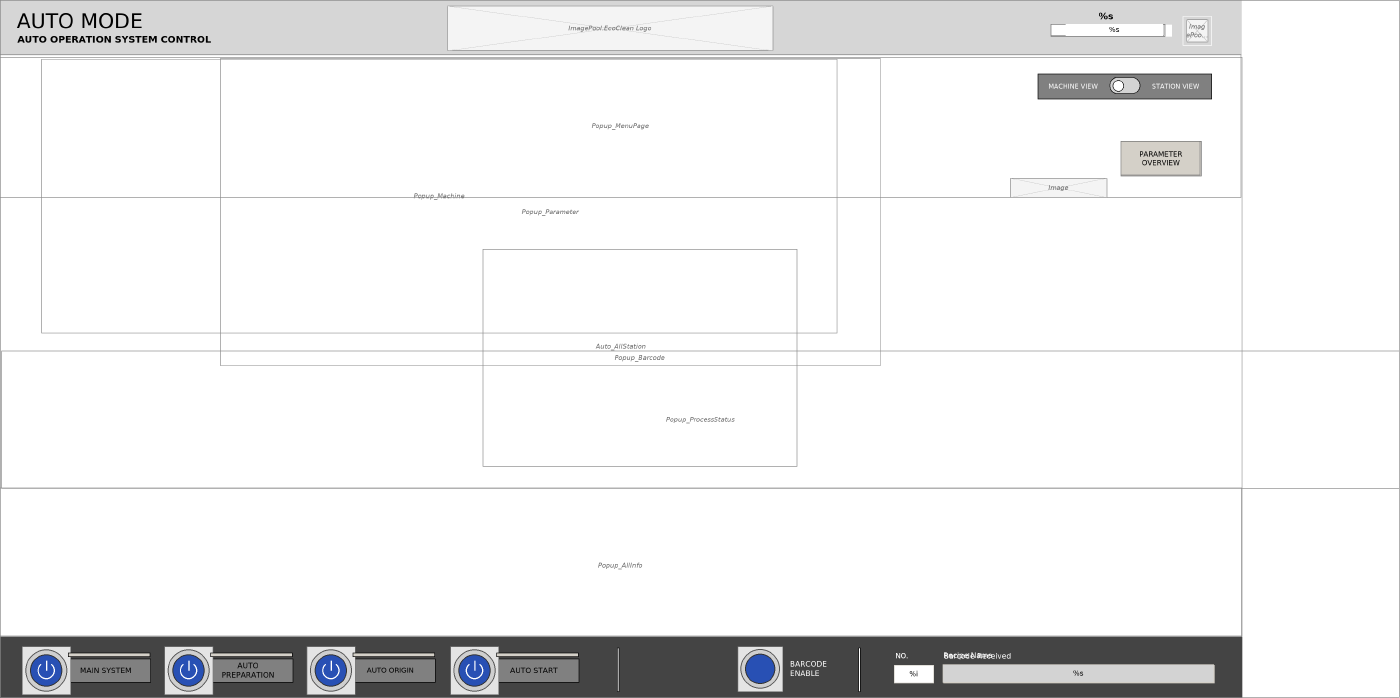
VISUALIZATION AutoMain_Page  // 2164x1079
    Rectangle (0,63 1920x26)
        p3528305787: HMI_Ctrl.ANIMATION3
    Rectangle (0,0 1919x85)
    Label (23,6 267x53), "AUTO MODE"
    Label (24,49 666x24), "AUTO OPERATION SYSTEM CONTROL"
    Frame (2,542 2161x213)
        shows Popup_ProcessStatus()
    Frame (-1,754 1920x240)
        shows Popup_AllInfo()
    Image (1561,275 150x30)
    Frame (64,91 1230x424)
        shows Popup_Machine()
    Group (1828,25 45x45)
        OnMouseClick: toggle HMI_Ctrl.MenuButton
        RoundedRectangle (0,0 45x45), colour toggle: HMI_Ctrl.MenuButton
        Image (6,5 33x35), image: ImagePool.Menu Button
    Group (1604,113 269x41), invisible if: HMI_Ctrl.AutoStationViewEnable
        RoundedRectangle (0,1 269x39)
        Label (1,0 108x41), "MACHINE VIEW"
        Label (161,0 105x41), "STATION VIEW"
        Group (111,6 47x26)
            OnMouseClick: toggle HMI_Ctrl.AutoStationViewEnable
            Group (0,0 47x26)
                Ellipse (0,0 26x26)
                Ellipse (21,0 26x26)
                RoundedRectangle (8,0 29x26)
            Ellipse (1,1 24x24)
            Ellipse (23,1 23x24)
            RoundedRectangle (9,1 28x24)
            Ellipse (5,5 17x17)
    Image (691,9 504x69), image: ImagePool.EcoClean Logo
    Rectangle (1661,38 150x18), "%s", text variable: fbHmiTF1800_UserlevelManagement.dsHmiUserStatus_Active.sLoginName
    Group (1621,14 180x42)
        Rectangle (0,0 177x22), "%s", text variable: DSLocalSystemTimeML.sCurrentDT24Hr_General
        Button (3,23 177x19), image: VisuSymbols.Symbols.AddUser
        Rectangle (26,23 150x18), "%s", text variable: fbHmiTF1800_UserlevelManagement.dsHmiUserStatus_Active.sLoginName
    Frame (340,90 1021x475), invisible if: NOT bParameterPopupPageOn
        shows Popup_Parameter()
    Frame (746,385 486x336), invisible if: NOT bAutoRecipeBarcodeCallPage
        shows Popup_Barcode()
    Button (1732,218 125x54), "PARAMETER OVERVIEW"
        toggle bParameterPopupPageOn
    Frame (0,88 1920x895), invisible if: NOT HMI_Ctrl.AutoStationViewEnable
        shows Auto_AllStation()
    Frame (0,84 1918x221), invisible if: HMI_Ctrl.CloseMenuButton
        shows Popup_MenuPage()
    Rectangle (0,984 1920x95)
    Group (1381,1002 496x54), invisible if: bBarcodeBypass
        Textfield (77,26 419x28), "%s", text variable: sBarcodeScannerReceivedCmd
        Label (0,0 62x24), "NO."
        Label (75,0 418x24), "Barcode Received"
        Textfield (1,26 61x28), "%i", text variable: HMI_Function.iRecipeNoFeed
    PushSwitch (1140,999 70x70), variable: bBarcodeEnable, behaviour: TOGGLE, style: Switch-PushSwitch-Blue
    Label (1218,1017 107x34), "BARCODE ENABLE"
    Rectangle (954,1001 3x68)
    Rectangle (1327,1001 3x68)
    RoundedRectangle (94,1018 139x37), "MAIN SYSTEM"
    PowerSwitch (34,999 75x75), variable: bMainOnOff, behaviour: TOGGLE, style: Switch-PowerSwitch-Blue
    RoundedRectangle (105,1009 127x6), colour toggle: bMainOnOff
    RoundedRectangle (314,1018 139x37), "AUTO PREPARATION"
    PowerSwitch (254,999 75x75), variable: bAutoPreparationPb, behaviour: TOGGLE, style: Switch-PowerSwitch-Blue
    RoundedRectangle (325,1009 127x6), colour toggle: bAutoPreparationDone
    RoundedRectangle (534,1018 139x37), "AUTO ORIGIN"
    PowerSwitch (474,999 75x75), variable: bAutoOriginPb, behaviour: TOGGLE, style: Switch-PowerSwitch-Blue
    RoundedRectangle (545,1009 127x6), colour toggle: bAutoOriginDone
    RoundedRectangle (756,1018 139x37), "AUTO START"
    PowerSwitch (696,999 75x75), variable: bAutoStartPb, behaviour: TOGGLE, style: Switch-PowerSwitch-Blue
    RoundedRectangle (767,1009 127x6), colour toggle: bAutoStartPb
    Group (1381,1001 495x55), invisible if: NOT bBarcodeBypass
        Label (0,1 50x24), "NO."
        Textfield (1,27 61x28), "%i", text variable: iUserDefineProductRecipeNo
            OnMouseDown: write the text variable via VisuDialogs.Numpad
        Textfield (76,26 419x28), "%s", text variable: ARsProductRecipeDescription[iUserDefineProductRecipeNo]
        Label (74,0 417x24), "Recipe Name"
END_VISUALIZATION

(* stored: Version 1.1.0.1, ProductVersion 3.1.4024.12
   Visu AutoMain_Page: Id {d1906453-8f43-4dd1-b197-c8b89271e837} *)
